FUNCTION_BLOCK FB_F_ValidateRequester_Test EXTENDS TcUnit.FB_TestSuite
VAR
END_VAR

AcceptsNormally();
AcceptsProgramWhenLocked();
RejectsOperatorWhenLocked();
SkipSourceCheckAllowsOperator();
RejectsWhenFaulted();
AcceptsWhenFaultedButAllowed();

METHOD AcceptsNormally
VAR
    nExpected : DINT := TcForge.E_RpcMethodResponse.ACCEPTED;
    nActual   : DINT;
END_VAR
TEST('AcceptsNormally');

nActual := TcForge.F_ValidateRequester(
    eRequester        := TcForge.E_Requester.OPERATOR,
    bSourceLocked     := FALSE,
    bFaulted          := FALSE,
    bAllowWhenFaulted := FALSE,
    bSkipSourceCheck  := FALSE);

AssertEquals_DINT(
    Expected := nExpected,
    Actual   := nActual,
    Message  := 'Should accept when there are no restrictions');

TEST_FINISHED();
END_METHOD

METHOD AcceptsProgramWhenLocked
VAR
    nExpected : DINT := TcForge.E_RpcMethodResponse.ACCEPTED;
    nActual   : DINT;
END_VAR
TEST('AcceptsProgramWhenLocked');

nActual := TcForge.F_ValidateRequester(
    eRequester        := TcForge.E_Requester.PROG,
    bSourceLocked     := TRUE,
    bFaulted          := FALSE,
    bAllowWhenFaulted := FALSE,
    bSkipSourceCheck  := FALSE);

AssertEquals_DINT(
    Expected := nExpected,
    Actual   := nActual,
    Message  := 'PROG requester should be accepted even when source is locked');

TEST_FINISHED();
END_METHOD

METHOD RejectsOperatorWhenLocked
VAR
    nExpected : DINT := TcForge.E_RpcMethodResponse.REJECTED_SOURCE_NOT_ALLOWED;
    nActual   : DINT;
END_VAR
TEST('RejectsOperatorWhenLocked');

nActual := TcForge.F_ValidateRequester(
    eRequester        := TcForge.E_Requester.OPERATOR,
    bSourceLocked     := TRUE,
    bFaulted          := FALSE,
    bAllowWhenFaulted := FALSE,
    bSkipSourceCheck  := FALSE);

AssertEquals_DINT(
    Expected := nExpected,
    Actual   := nActual,
    Message  := 'OPERATOR must be rejected when source is locked');

TEST_FINISHED();
END_METHOD

METHOD SkipSourceCheckAllowsOperator
VAR
    nExpected : DINT := TcForge.E_RpcMethodResponse.ACCEPTED;
    nActual   : DINT;
END_VAR
TEST('SkipSourceCheckAllowsOperator');

nActual := TcForge.F_ValidateRequester(
    eRequester        := TcForge.E_Requester.OPERATOR,
    bSourceLocked     := TRUE,
    bFaulted          := FALSE,
    bAllowWhenFaulted := FALSE,
    bSkipSourceCheck  := TRUE);

AssertEquals_DINT(
    Expected := nExpected,
    Actual   := nActual,
    Message  := 'bSkipSourceCheck should bypass the lock and accept OPERATOR');

TEST_FINISHED();
END_METHOD

METHOD RejectsWhenFaulted
VAR
    nExpected : DINT := TcForge.E_RpcMethodResponse.REJECTED_FAULTED;
    nActual   : DINT;
END_VAR
TEST('RejectsWhenFaulted');

nActual := TcForge.F_ValidateRequester(
    eRequester        := TcForge.E_Requester.OPERATOR,
    bSourceLocked     := FALSE,
    bFaulted          := TRUE,
    bAllowWhenFaulted := FALSE,
    bSkipSourceCheck  := FALSE);

AssertEquals_DINT(
    Expected := nExpected,
    Actual   := nActual,
    Message  := 'Should reject when faulted and bAllowWhenFaulted is FALSE');

TEST_FINISHED();
END_METHOD

METHOD AcceptsWhenFaultedButAllowed
VAR
    nExpected : DINT := TcForge.E_RpcMethodResponse.ACCEPTED;
    nActual   : DINT;
END_VAR
TEST('AcceptsWhenFaultedButAllowed');

nActual := TcForge.F_ValidateRequester(
    eRequester        := TcForge.E_Requester.OPERATOR,
    bSourceLocked     := FALSE,
    bFaulted          := TRUE,
    bAllowWhenFaulted := TRUE,
    bSkipSourceCheck  := FALSE);

AssertEquals_DINT(
    Expected := nExpected,
    Actual   := nActual,
    Message  := 'Should accept when faulted but bAllowWhenFaulted is TRUE');

TEST_FINISHED();
END_METHOD

END_FUNCTION_BLOCK

(* stored: Version 1.1.0.1, ProductVersion 3.1.4026.12
   POU FB_F_ValidateRequester_Test: Id {a1b2c3d4-e5f6-7890-abcd-ef1234560001}, SpecialFunc None
   Method AcceptsNormally: Id {a1b2c3d4-e5f6-7890-abcd-ef1234560002}
   Method AcceptsProgramWhenLocked: Id {a1b2c3d4-e5f6-7890-abcd-ef1234560003}
   Method RejectsOperatorWhenLocked: Id {a1b2c3d4-e5f6-7890-abcd-ef1234560004}
   Method SkipSourceCheckAllowsOperator: Id {a1b2c3d4-e5f6-7890-abcd-ef1234560005}
   Method RejectsWhenFaulted: Id {a1b2c3d4-e5f6-7890-abcd-ef1234560006}
   Method AcceptsWhenFaultedButAllowed: Id {a1b2c3d4-e5f6-7890-abcd-ef1234560007} *)
